PROGRAM pouStation1Motions
VAR
	row1: FB_HMI_Control;
	row2: FB_HMI_Control;
	row3: FB_HMI_Control;
	row4: FB_HMI_Control;
	row5: FB_HMI_Control;
	row6: FB_HMI_Control;
	row7: FB_HMI_Control;
	row8: FB_HMI_Control;
	row9: FB_HMI_Control;
	row10: FB_HMI_Control;
	tNumberOfPages: REAL;
	tCalcNumberOfPages: REAL;
	row11: FB_HMI_Control;
	row12: FB_HMI_Control;
	row13: FB_HMI_Control;
	row14: FB_HMI_Control;
	row15: FB_HMI_Control;
	row16: FB_HMI_Control;
	row17: FB_HMI_Control;
	row18: FB_HMI_Control;
	row19: FB_HMI_Control;
	row20: FB_HMI_Control;
	row21: FB_HMI_Control;
	row22: FB_HMI_Control;
	row23: FB_HMI_Control;
	row24: FB_HMI_Control;
	//StationNativeMotionRows: ARRAY[0..99] OF typeMotionRow;
	ceil: LREAL;
END_VAR

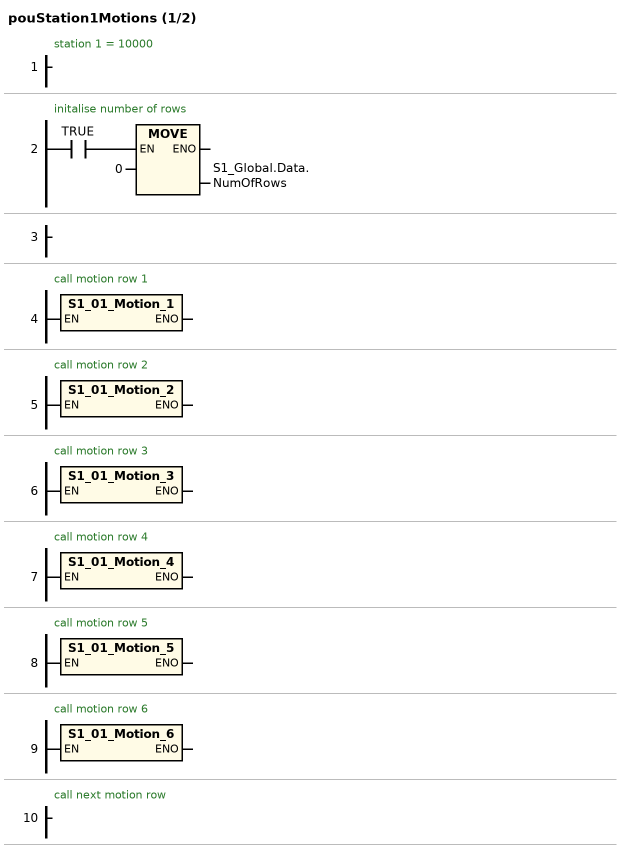
// NETWORK 1
// station 1 = 10000

// NETWORK 2
// initalise number of rows
S1_Global.Data.NumOfRows := 0;

// NETWORK 3

// NETWORK 4
// call motion row 1
S1_01_Motion_1();

// NETWORK 5
// call motion row 2
S1_01_Motion_2();

// NETWORK 6
// call motion row 3
S1_01_Motion_3();

// NETWORK 7
// call motion row 4
S1_01_Motion_4();

// NETWORK 8
// call motion row 5
S1_01_Motion_5();

// NETWORK 9
// call motion row 6
S1_01_Motion_6();

// NETWORK 10
// call next motion row

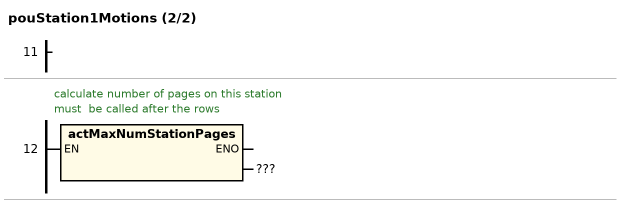
// NETWORK 11

// NETWORK 12
// calculate number of pages on this station
// must  be called after the rows
actMaxNumStationPages();

ACTION actMaxNumStationPages:
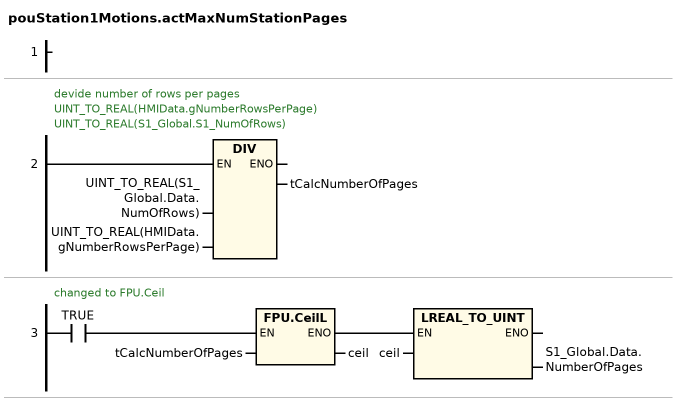
// NETWORK 1

// NETWORK 2
// devide number of rows per pages
// UINT_TO_REAL(HMIData.gNumberRowsPerPage)
// UINT_TO_REAL(S1_Global.S1_NumOfRows)
tCalcNumberOfPages := (UINT_TO_REAL(S1_Global.Data.NumOfRows)) / (UINT_TO_REAL(HMIData.gNumberRowsPerPage));

// NETWORK 3
// changed to FPU.Ceil
ceil := FPU.CeilL(tCalcNumberOfPages);
S1_Global.Data.NumberOfPages := LREAL_TO_UINT(ceil);
END_ACTION

END_PROGRAM

(* stored: Version 1.1.0.1, ProductVersion 3.1.4024.12
   POU pouStation1Motions: Id {c7fc4120-0f64-4600-a362-aff930f91025}, SpecialFunc None
   Action actMaxNumStationPages: Id {499acf2e-11f1-41ab-acd8-6d6b219bcc13} *)
